FUNCTION_BLOCK TRAIN_TEST_SPLIT_FB
  {SET_ATTRIBUTE(OpcUa, SERVICE)}
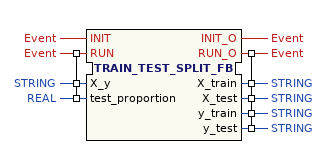
  EVENT_INPUT
    INIT;
    RUN WITH X_y, test_proportion; {SET_ATTRIBUTE(OpcUa, Method)}
  END_EVENT
  EVENT_OUTPUT
    INIT_O;
    RUN_O WITH X_train, X_test, y_train, y_test;
  END_EVENT
  VAR_INPUT
    X_y : STRING; {SET_ATTRIBUTE(OpcUa, Variable.RUN)}
    test_proportion : REAL; {SET_ATTRIBUTE(OpcUa, Variable.RUN)}
  END_VAR
  VAR_OUTPUT
    X_train : STRING; {SET_ATTRIBUTE(OpcUa, Variable.RUN)}
    X_test : STRING; {SET_ATTRIBUTE(OpcUa, Variable.RUN)}
    y_train : STRING; {SET_ATTRIBUTE(OpcUa, Variable.RUN)}
    y_test : STRING; {SET_ATTRIBUTE(OpcUa, Variable.RUN)}
  END_VAR
END_FUNCTION_BLOCK
